Omron Sysmac Studio project oen_library_mqtt_nx1p2 (Sysmac Studio 1.45.1.64010, StandardProject)

# Controller new_Controller_0: NX1P2-9024DT version 1.40
Task PrimaryTask (priority 4, period or condition 2000): Program0
Library OEN_BaseBlocks 5.00 5.00.10 (contents left out)
Library OEN_Communication_V1_0_22 1.0.22 (contents left out)
Library OEN_Components 1.06.5 (contents left out)
Library OmronLib_MQTT_Comm_V1_0 1.0.0 (contents left out)
Library JSON 0.0.55 (contents left out)

PROGRAM Program0
VAR
    fist_runmode : BOOL;
    connect_setting_mqtt : OmronLib\MQTT_Comm\MQTTClient;
    connect_setting_local : OmronLib\MQTT_Comm\sConnectionSettings;
    Pup_topic : STRING[256];
    pub_pubsetting_pubOs : WORD;
    pub_pubsetting_RetainFlag : BOOL;
    Sub_topic : STRING[256];
    connect : BOOL;
    FB_MQTT_CLIENT_LOCAL : OmronLib\MQTT_Comm\MQTTClient;
    CLIENT_REFERRENCE_LOCAL : OmronLib\MQTT_Comm\sClientReference;
    fb_mqtt_substring : OmronLib\MQTT_Comm\MQTTPubString;
    pub_packetID : UINT;
    pub_msgtype : USINT;
    pub_msg : STRING[1986];
    pub_setting : OmronLib\MQTT_Comm\sPubFlags;
    pub_topic : STRING[512];
END_VAR

(* Section mqtt_local: ladder, written here as Structured Text *)

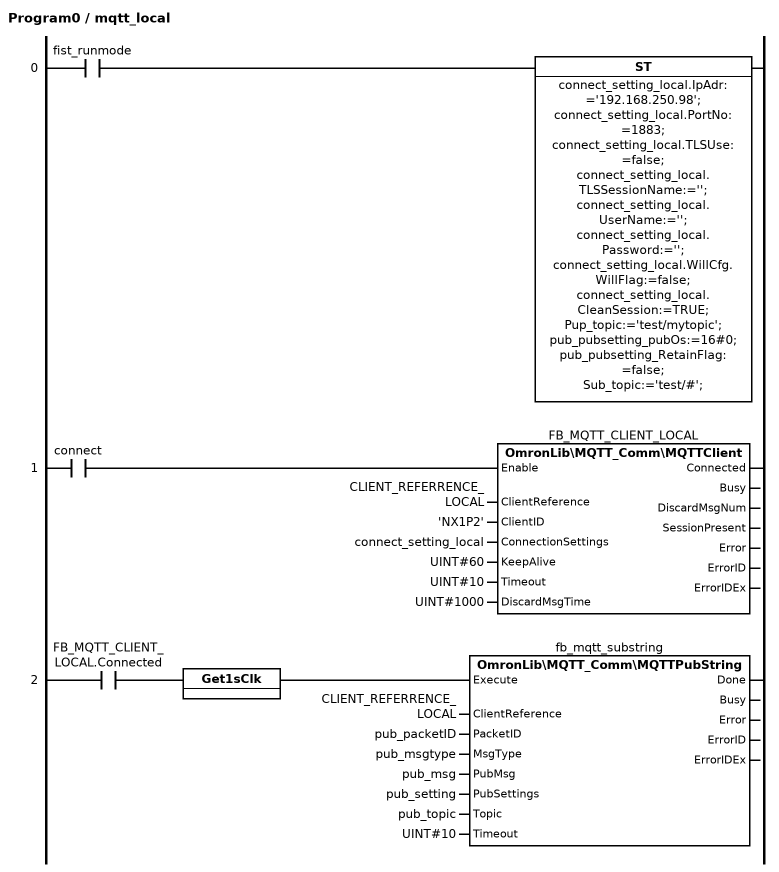
(* Rung 0 *)
IF fist_runmode THEN
    connect_setting_local.IpAdr:='192.168.250.98';
    connect_setting_local.PortNo:=1883;
    connect_setting_local.TLSUse:=false;
    connect_setting_local.TLSSessionName:='';
    connect_setting_local.UserName:='';
    connect_setting_local.Password:='';
    connect_setting_local.WillCfg.WillFlag:=false;
    connect_setting_local.CleanSession:=TRUE;
    
    Pup_topic:='test/mytopic';
    
    pub_pubsetting_pubOs:=16#0;
    pub_pubsetting_RetainFlag:=false;
    
    Sub_topic:='test/#';
END_IF;
(* Rung 1 *)
FB_MQTT_CLIENT_LOCAL(Enable := connect, ClientReference := CLIENT_REFERRENCE_LOCAL, ClientID := 'NX1P2', ConnectionSettings := connect_setting_local, KeepAlive := UINT#60, Timeout := UINT#10, DiscardMsgTime := UINT#1000);
(* Rung 2 *)
fb_mqtt_substring(Execute := FB_MQTT_CLIENT_LOCAL.Connected AND Get1sClk(), ClientReference := CLIENT_REFERRENCE_LOCAL, PacketID := pub_packetID, MsgType := pub_msgtype, PubMsg := pub_msg, PubSettings := pub_setting, Topic := pub_topic, Timeout := UINT#10);
END_PROGRAM